TYPE ST_HE_SolidAttenuatorSettings :
STRUCT
    bEnabled : BOOL;
    eMode : E_HE_SolidAttenuatorCalculationMode;
    bDynamicCalculation : BOOL;
END_STRUCT
END_TYPE

(* stored: Version 1.1.0.1
   DUT ST_HE_SolidAttenuatorSettings: Id {147303cb-e30a-4a5b-9079-8e5e4423f267} *)
